(* IEC 61131-3 sources: Fischertechnik-RPi/Test, 12 files *)

(* ---- 1test.st ---- *)
PROGRAM Cell1
  VAR
    R1_front AT %IX0.2 : BOOL := true;
    R1_rear AT %IX0.3 : BOOL := true;
    C1_endIR AT %IX0.4 : BOOL := true;
    C1_startIR AT %IX0.5 : BOOL := true;
    Main AT %IX0.6 : BOOL := false;
    R1_fwd_motor AT %QX0.2 : BOOL := true;
    R1_bwd_motor AT %QX0.3 : BOOL := true;
    C1_motor AT %QX0.4 : BOOL := true;
  END_VAR
  VAR
    C1_working : BOOL := false;
    State1 : BOOL := false;
  END_VAR
  VAR
    State1_int AT %MD1 : DINT := 0;
  END_VAR
  VAR
    R1_in_transit : BOOL := false;
    State2 : BOOL := false;
  END_VAR
  VAR
    State2_int AT %MD3 : DINT := 0;
  END_VAR
  VAR
    R1_fwd : BOOL := false;
  END_VAR
  VAR
    R1_fwd_int AT %MD4 : DINT := 0;
  END_VAR
  VAR
    R1_bwd : BOOL := false;
  END_VAR
  VAR
    R1_bwd_int AT %MD5 : DINT := 0;
  END_VAR
  VAR
    Timer_in_transit : TON;
    BOOL_TO_DINT27_ENO : BOOL;
    BOOL_TO_DINT27_OUT : DINT;
    BOOL_TO_DINT37_ENO : BOOL;
    BOOL_TO_DINT37_OUT : DINT;
    BOOL_TO_DINT61_ENO : BOOL;
    BOOL_TO_DINT61_OUT : DINT;
    BOOL_TO_DINT67_ENO : BOOL;
    BOOL_TO_DINT67_OUT : DINT;
  END_VAR

  IF NOT(C1_startIR) THEN
    C1_working := TRUE; (*set*)
  END_IF;
  C1_motor := NOT(C1_working AND NOT(Main));
  IF C1_working AND NOT(C1_endIR) THEN
    R1_in_transit := TRUE; (*set*)
  END_IF;
  Timer_in_transit(IN := R1_in_transit AND C1_working, PT := T#1000ms);
  IF Timer_in_transit.Q THEN
    R1_fwd := TRUE; (*set*)
  END_IF;
  IF Timer_in_transit.Q THEN
    C1_working := FALSE; (*reset*)
  END_IF;
  IF Timer_in_transit.Q THEN
    R1_in_transit := FALSE; (*reset*)
  END_IF;
  R1_fwd_motor := NOT(R1_fwd AND NOT(Main));
  IF NOT(R1_front) AND R1_fwd THEN
    R1_bwd := TRUE; (*set*)
  END_IF;
  IF NOT(R1_front) AND R1_fwd THEN
    R1_fwd := FALSE; (*reset*)
  END_IF;
  R1_bwd_motor := NOT(R1_bwd AND NOT(Main));
  IF NOT(R1_rear) AND R1_bwd THEN
    R1_bwd := FALSE; (*reset*)
  END_IF;
  IF R1_in_transit AND C1_working THEN
    State1 := FALSE; (*reset*)
  END_IF;
  IF R1_in_transit AND C1_working THEN
    State2 := TRUE; (*set*)
  END_IF;
  IF NOT(R1_in_transit) AND C1_working THEN
    State1 := TRUE; (*set*)
  END_IF;
  IF NOT(R1_in_transit) AND NOT(C1_working) THEN
    State2 := FALSE; (*reset*)
  END_IF;
  BOOL_TO_DINT27_OUT := BOOL_TO_DINT(EN := TRUE, IN := State1, ENO => BOOL_TO_DINT27_ENO);
  State1_int := BOOL_TO_DINT27_OUT;
  BOOL_TO_DINT37_OUT := BOOL_TO_DINT(EN := TRUE, IN := State2, ENO => BOOL_TO_DINT37_ENO);
  State2_int := BOOL_TO_DINT37_OUT;
  BOOL_TO_DINT61_OUT := BOOL_TO_DINT(EN := TRUE, IN := R1_fwd, ENO => BOOL_TO_DINT61_ENO);
  R1_fwd_int := BOOL_TO_DINT61_OUT;
  BOOL_TO_DINT67_OUT := BOOL_TO_DINT(EN := TRUE, IN := R1_bwd, ENO => BOOL_TO_DINT67_ENO);
  R1_bwd_int := BOOL_TO_DINT67_OUT;
END_PROGRAM

CONFIGURATION Config0

  RESOURCE Res0 ON PLC
    TASK TaskMain(INTERVAL := T#50ms,PRIORITY := 0);
    PROGRAM Inst0 WITH TaskMain : Cell1;
  END_RESOURCE
END_CONFIGURATION

(* ---- FT_con02.st ---- *)
PROGRAM Cell2
  VAR
    C1_IR AT %IX0.3 : BOOL := true;
    M1_IR AT %IX0.4 : BOOL := true;
    Main AT %IX0.6 : BOOL := true;
    M1_motor AT %QX0.2 : BOOL := true;
    C2_motor AT %QX0.4 : BOOL := true;
  END_VAR
  VAR
    C2_working : BOOL := false;
  END_VAR
  VAR
    C2_working_int AT %MD1 : DINT := 0;
  END_VAR
  VAR
    C2_afterM : BOOL := false;
  END_VAR
  VAR
    C2_afterM_int AT %MD2 : DINT := 0;
  END_VAR
  VAR
    Step1 : BOOL := false;
  END_VAR
  VAR
    Step1_int AT %MD3 : DINT := 0;
  END_VAR
  VAR
    Step2 : BOOL := false;
  END_VAR
  VAR
    Step2_int AT %MD4 : DINT := 0;
  END_VAR
  VAR
    Step3 : BOOL := false;
  END_VAR
  VAR
    Step3_int AT %MD5 : DINT := 0;
  END_VAR
  VAR
    Pause1 : BOOL := false;
  END_VAR
  VAR
    Pause1_int AT %MD6 : DINT := 0;
  END_VAR
  VAR
    Pause2 : BOOL := false;
  END_VAR
  VAR
    Pause2_int AT %MD7 : DINT := 0;
  END_VAR
  VAR
    Timer_conveyor : TON;
    Timer_machining : TON;
    TON0 : TON;
    TON1 : TON;
    TON2 : TON;
    TON3 : TON;
    TON4 : TON;
    BOOL_TO_DINT41_ENO : BOOL;
    BOOL_TO_DINT41_OUT : DINT;
    BOOL_TO_DINT105_ENO : BOOL;
    BOOL_TO_DINT105_OUT : DINT;
    BOOL_TO_DINT51_ENO : BOOL;
    BOOL_TO_DINT51_OUT : DINT;
    BOOL_TO_DINT85_ENO : BOOL;
    BOOL_TO_DINT85_OUT : DINT;
    BOOL_TO_DINT90_ENO : BOOL;
    BOOL_TO_DINT90_OUT : DINT;
    BOOL_TO_DINT95_ENO : BOOL;
    BOOL_TO_DINT95_OUT : DINT;
    BOOL_TO_DINT100_ENO : BOOL;
    BOOL_TO_DINT100_OUT : DINT;
  END_VAR

  IF NOT(C1_IR) THEN
    C2_working := TRUE; (*set*)
  END_IF;
  C2_motor := NOT((C2_afterM OR C2_working) AND NOT(Main));
  IF NOT(M1_IR) AND C2_working THEN
    Step1 := TRUE; (*set*)
  END_IF;
  IF NOT(M1_IR) AND C2_working THEN
    C2_working := FALSE; (*reset*)
  END_IF;
  M1_motor := NOT((Step1 OR Step2 OR Step3) AND NOT(Main));
  TON0(IN := Step1, PT := T#1000ms);
  IF TON0.Q THEN
    Pause1 := TRUE; (*set*)
  END_IF;
  IF TON0.Q THEN
    Step1 := FALSE; (*reset*)
  END_IF;
  TON1(IN := Pause1, PT := T#1000ms);
  IF TON1.Q THEN
    Pause1 := FALSE; (*reset*)
  END_IF;
  IF TON1.Q THEN
    Step2 := TRUE; (*set*)
  END_IF;
  TON2(IN := Step2, PT := T#1000ms);
  IF TON2.Q THEN
    Pause2 := TRUE; (*set*)
  END_IF;
  IF TON2.Q THEN
    Step2 := FALSE; (*reset*)
  END_IF;
  TON3(IN := Pause2, PT := T#1000ms);
  IF TON3.Q THEN
    Pause2 := FALSE; (*reset*)
  END_IF;
  IF TON3.Q THEN
    Step3 := TRUE; (*set*)
  END_IF;
  Timer_machining(IN := Step3, PT := T#1000ms);
  IF Timer_machining.Q THEN
    C2_afterM := TRUE; (*set*)
  END_IF;
  IF Timer_machining.Q THEN
    Step3 := FALSE; (*reset*)
  END_IF;
  Timer_conveyor(IN := C2_working, PT := T#6000ms);
  IF Timer_conveyor.Q THEN
    C2_working := FALSE; (*reset*)
  END_IF;
  TON4(IN := C2_afterM, PT := T#2000ms);
  IF TON4.Q THEN
    C2_afterM := FALSE; (*reset*)
  END_IF;
  BOOL_TO_DINT41_OUT := BOOL_TO_DINT(EN := TRUE, IN := C2_working, ENO => BOOL_TO_DINT41_ENO);
  C2_working_int := BOOL_TO_DINT41_OUT;
  BOOL_TO_DINT105_OUT := BOOL_TO_DINT(EN := TRUE, IN := C2_afterM, ENO => BOOL_TO_DINT105_ENO);
  C2_afterM_int := BOOL_TO_DINT105_OUT;
  BOOL_TO_DINT51_OUT := BOOL_TO_DINT(EN := TRUE, IN := Step1, ENO => BOOL_TO_DINT51_ENO);
  Step1_int := BOOL_TO_DINT51_OUT;
  BOOL_TO_DINT85_OUT := BOOL_TO_DINT(EN := TRUE, IN := Step2, ENO => BOOL_TO_DINT85_ENO);
  Step2_int := BOOL_TO_DINT85_OUT;
  BOOL_TO_DINT90_OUT := BOOL_TO_DINT(EN := TRUE, IN := Step3, ENO => BOOL_TO_DINT90_ENO);
  Step3_int := BOOL_TO_DINT90_OUT;
  BOOL_TO_DINT95_OUT := BOOL_TO_DINT(EN := TRUE, IN := Pause1, ENO => BOOL_TO_DINT95_ENO);
  Pause1_int := BOOL_TO_DINT95_OUT;
  BOOL_TO_DINT100_OUT := BOOL_TO_DINT(EN := TRUE, IN := Pause2, ENO => BOOL_TO_DINT100_ENO);
  Pause2_int := BOOL_TO_DINT100_OUT;
END_PROGRAM

CONFIGURATION Config0

  RESOURCE Res0 ON PLC
    TASK TaskMain(INTERVAL := T#50ms,PRIORITY := 0);
    PROGRAM Inst0 WITH TaskMain : Cell2;
  END_RESOURCE
END_CONFIGURATION

(* ---- FT_con03.st ---- *)
PROGRAM Cell3
  VAR
    C2_IR AT %IX0.3 : BOOL := true;
    M2_IR AT %IX0.4 : BOOL := true;
    Main AT %IX0.6 : BOOL := true;
    M2_motor AT %QX0.2 : BOOL := true;
    C3_motor AT %QX0.4 : BOOL := true;
  END_VAR
  VAR
    C3_working : BOOL := false;
  END_VAR
  VAR
    C3_working_int AT %MD1 : DINT := 0;
  END_VAR
  VAR
    C3_afterM : BOOL := false;
  END_VAR
  VAR
    C3_afterM_int AT %MD2 : DINT := 0;
  END_VAR
  VAR
    Step1 : BOOL := false;
  END_VAR
  VAR
    Step1_int AT %MD3 : DINT := 0;
  END_VAR
  VAR
    Step2 : BOOL := false;
  END_VAR
  VAR
    Step2_int AT %MD4 : DINT := 0;
  END_VAR
  VAR
    Pause : BOOL := false;
  END_VAR
  VAR
    Pause_int AT %MD5 : DINT := 0;
  END_VAR
  VAR
    Timer_conveyor : TON;
    Timer_machining : TON;
    TON0 : TON;
    TON1 : TON;
    TON2 : TON;
    TON3 : TON;
    BOOL_TO_DINT70_ENO : BOOL;
    BOOL_TO_DINT70_OUT : DINT;
    BOOL_TO_DINT41_ENO : BOOL;
    BOOL_TO_DINT41_OUT : DINT;
    BOOL_TO_DINT51_ENO : BOOL;
    BOOL_TO_DINT51_OUT : DINT;
    BOOL_TO_DINT75_ENO : BOOL;
    BOOL_TO_DINT75_OUT : DINT;
    BOOL_TO_DINT80_ENO : BOOL;
    BOOL_TO_DINT80_OUT : DINT;
  END_VAR

  TON0(IN := NOT(C2_IR), PT := T#5000ms);
  IF TON0.Q THEN
    C3_working := TRUE; (*set*)
  END_IF;
  C3_motor := NOT((C3_afterM OR C3_working) AND NOT(Main));
  IF NOT(M2_IR) AND C3_working THEN
    Step1 := TRUE; (*set*)
  END_IF;
  IF NOT(M2_IR) AND C3_working THEN
    C3_working := FALSE; (*reset*)
  END_IF;
  M2_motor := NOT((Step1 OR Step2) AND NOT(Main));
  Timer_machining(IN := Step1, PT := T#2000ms);
  IF Timer_machining.Q THEN
    Pause := TRUE; (*set*)
  END_IF;
  IF Timer_machining.Q THEN
    Step1 := FALSE; (*reset*)
  END_IF;
  TON2(IN := Pause, PT := T#1000ms);
  IF TON2.Q THEN
    Step2 := TRUE; (*set*)
  END_IF;
  IF TON2.Q THEN
    Pause := FALSE; (*reset*)
  END_IF;
  TON1(IN := Step2, PT := T#2000ms);
  IF TON1.Q THEN
    C3_afterM := TRUE; (*set*)
  END_IF;
  IF TON1.Q THEN
    Step2 := FALSE; (*reset*)
  END_IF;
  Timer_conveyor(IN := C3_working, PT := T#6000ms);
  IF Timer_conveyor.Q THEN
    C3_working := FALSE; (*reset*)
  END_IF;
  TON3(IN := C3_afterM, PT := T#3000ms);
  IF TON3.Q THEN
    C3_afterM := FALSE; (*reset*)
  END_IF;
  BOOL_TO_DINT70_OUT := BOOL_TO_DINT(EN := TRUE, IN := C3_working, ENO => BOOL_TO_DINT70_ENO);
  C3_working_int := BOOL_TO_DINT70_OUT;
  BOOL_TO_DINT41_OUT := BOOL_TO_DINT(EN := TRUE, IN := C3_afterM, ENO => BOOL_TO_DINT41_ENO);
  C3_afterM_int := BOOL_TO_DINT41_OUT;
  BOOL_TO_DINT51_OUT := BOOL_TO_DINT(EN := TRUE, IN := Step1, ENO => BOOL_TO_DINT51_ENO);
  Step1_int := BOOL_TO_DINT51_OUT;
  BOOL_TO_DINT75_OUT := BOOL_TO_DINT(EN := TRUE, IN := Step2, ENO => BOOL_TO_DINT75_ENO);
  Step2_int := BOOL_TO_DINT75_OUT;
  BOOL_TO_DINT80_OUT := BOOL_TO_DINT(EN := TRUE, IN := Pause, ENO => BOOL_TO_DINT80_ENO);
  Pause_int := BOOL_TO_DINT80_OUT;
END_PROGRAM

CONFIGURATION Config0

  RESOURCE Res0 ON PLC
    TASK TaskMain(INTERVAL := T#50ms,PRIORITY := 0);
    PROGRAM Inst0 WITH TaskMain : Cell3;
  END_RESOURCE
END_CONFIGURATION

(* ---- FT_con04.st ---- *)
PROGRAM Cell4
  VAR
    R2_front AT %IX0.2 : BOOL := true;
    R2_rear AT %IX0.3 : BOOL := true;
    C4_endIR AT %IX0.4 : BOOL := true;
    C3_IR AT %IX0.5 : BOOL := true;
    Main AT %IX0.6 : BOOL := false;
    R2_fwd_motor AT %QX0.2 : BOOL := true;
    R2_bwd_motor AT %QX0.3 : BOOL := true;
    C4_motor AT %QX0.4 : BOOL := true;
  END_VAR
  VAR
    C4_working : BOOL := false;
  END_VAR
  VAR
    C4_working_int AT %MD1 : DINT := 0;
  END_VAR
  VAR
    R2_in_transit : BOOL := false;
  END_VAR
  VAR
    R2_in_transit_int AT %MD3 : DINT := 0;
  END_VAR
  VAR
    R2_fwd : BOOL := false;
  END_VAR
  VAR
    R2_fwd_int AT %MD4 : DINT := 0;
  END_VAR
  VAR
    R2_bwd : BOOL := false;
  END_VAR
  VAR
    R2_bwd_int AT %MD5 : DINT := 0;
  END_VAR
  VAR
    Timer_in_transit : TON;
    BOOL_TO_DINT49_ENO : BOOL;
    BOOL_TO_DINT49_OUT : DINT;
    BOOL_TO_DINT64_ENO : BOOL;
    BOOL_TO_DINT64_OUT : DINT;
    BOOL_TO_DINT61_ENO : BOOL;
    BOOL_TO_DINT61_OUT : DINT;
    BOOL_TO_DINT67_ENO : BOOL;
    BOOL_TO_DINT67_OUT : DINT;
  END_VAR

  IF NOT(C3_IR) THEN
    R2_in_transit := TRUE; (*set*)
  END_IF;
  Timer_in_transit(IN := R2_in_transit, PT := T#6000ms);
  IF Timer_in_transit.Q THEN
    R2_fwd := TRUE; (*set*)
  END_IF;
  IF Timer_in_transit.Q THEN
    C4_working := TRUE; (*set*)
  END_IF;
  IF Timer_in_transit.Q THEN
    R2_in_transit := FALSE; (*reset*)
  END_IF;
  R2_fwd_motor := NOT(R2_fwd AND NOT(Main));
  IF NOT(R2_front) AND R2_fwd THEN
    R2_bwd := TRUE; (*set*)
  END_IF;
  IF NOT(R2_front) AND R2_fwd THEN
    R2_fwd := FALSE; (*reset*)
  END_IF;
  R2_bwd_motor := NOT(R2_bwd AND NOT(Main) AND TRUE);
  IF NOT(R2_rear) AND R2_bwd THEN
    R2_bwd := FALSE; (*reset*)
  END_IF;
  C4_motor := NOT(C4_working AND NOT(Main));
  IF NOT(C4_endIR) AND C4_working THEN
    C4_working := FALSE; (*reset*)
  END_IF;
  BOOL_TO_DINT49_OUT := BOOL_TO_DINT(EN := TRUE, IN := C4_working, ENO => BOOL_TO_DINT49_ENO);
  C4_working_int := BOOL_TO_DINT49_OUT;
  BOOL_TO_DINT64_OUT := BOOL_TO_DINT(EN := TRUE, IN := R2_in_transit, ENO => BOOL_TO_DINT64_ENO);
  R2_in_transit_int := BOOL_TO_DINT64_OUT;
  BOOL_TO_DINT61_OUT := BOOL_TO_DINT(EN := TRUE, IN := R2_fwd, ENO => BOOL_TO_DINT61_ENO);
  R2_fwd_int := BOOL_TO_DINT61_OUT;
  BOOL_TO_DINT67_OUT := BOOL_TO_DINT(EN := TRUE, IN := R2_bwd, ENO => BOOL_TO_DINT67_ENO);
  R2_bwd_int := BOOL_TO_DINT67_OUT;
END_PROGRAM

CONFIGURATION Config0

  RESOURCE Res0 ON PLC
    TASK TaskMain(INTERVAL := T#50ms,PRIORITY := 0);
    PROGRAM Inst0 WITH TaskMain : Cell4;
  END_RESOURCE
END_CONFIGURATION

(* ---- FT_con04b.st ---- *)
PROGRAM Cell4
  VAR
    R2_front AT %IX0.2 : BOOL := true;
    R2_rear AT %IX0.3 : BOOL := true;
    C4_endIR AT %IX0.4 : BOOL := true;
    C3_IR AT %IX0.5 : BOOL := true;
    Main AT %IX0.6 : BOOL := false;
    R2_fwd_motor AT %QX0.2 : BOOL := true;
    R2_bwd_motor AT %QX0.3 : BOOL := true;
    C4_motor AT %QX0.4 : BOOL := true;
  END_VAR
  VAR
    C4_working : BOOL := false;
    C4_R2f : BOOL := false;
  END_VAR
  VAR
    C4_R2f_int AT %MD1 : DINT := 0;
  END_VAR
  VAR
    R2_in_transit : BOOL := false;
  END_VAR
  VAR
    R2_in_transit_int AT %MD3 : DINT := 0;
  END_VAR
  VAR
    R2_fwd : BOOL := false;
    C4_R2b : BOOL := false;
  END_VAR
  VAR
    C4_R2b_int AT %MD4 : DINT := 0;
  END_VAR
  VAR
    R2_bwd : BOOL := false;
    R2b_solo : BOOL := false;
  END_VAR
  VAR
    R2b_solo_int AT %MD5 : DINT := 0;
  END_VAR
  VAR
    Timer_in_transit : TON;
    BOOL_TO_DINT49_ENO : BOOL;
    BOOL_TO_DINT49_OUT : DINT;
    BOOL_TO_DINT64_ENO : BOOL;
    BOOL_TO_DINT64_OUT : DINT;
    BOOL_TO_DINT61_ENO : BOOL;
    BOOL_TO_DINT61_OUT : DINT;
    BOOL_TO_DINT67_ENO : BOOL;
    BOOL_TO_DINT67_OUT : DINT;
  END_VAR

  IF NOT(C3_IR) THEN
    R2_in_transit := TRUE; (*set*)
  END_IF;
  Timer_in_transit(IN := R2_in_transit, PT := T#6000ms);
  IF Timer_in_transit.Q THEN
    R2_fwd := TRUE; (*set*)
  END_IF;
  IF Timer_in_transit.Q THEN
    C4_working := TRUE; (*set*)
  END_IF;
  IF Timer_in_transit.Q THEN
    R2_in_transit := FALSE; (*reset*)
  END_IF;
  R2_fwd_motor := NOT(R2_fwd AND NOT(Main));
  IF NOT(R2_front) AND R2_fwd THEN
    R2_bwd := TRUE; (*set*)
  END_IF;
  IF NOT(R2_front) AND R2_fwd THEN
    R2_fwd := FALSE; (*reset*)
  END_IF;
  R2_bwd_motor := NOT(R2_bwd AND NOT(Main) AND TRUE);
  IF NOT(R2_rear) AND R2_bwd THEN
    R2_bwd := FALSE; (*reset*)
  END_IF;
  IF NOT(R2_bwd) THEN
    R2b_solo := FALSE; (*reset*)
  END_IF;
  C4_motor := NOT(C4_working AND NOT(Main));
  IF NOT(C4_endIR) AND C4_working THEN
    C4_working := FALSE; (*reset*)
  END_IF;
  IF R2_fwd AND C4_working THEN
    C4_R2f := TRUE; (*set*)
  END_IF;
  IF R2_bwd AND C4_working THEN
    C4_R2b := TRUE; (*set*)
  END_IF;
  IF R2_fwd AND C4_working THEN
    C4_R2f := TRUE; (*set*)
  END_IF;
  IF R2_fwd AND C4_working THEN
    C4_R2f := TRUE; (*set*)
  END_IF;
  IF R2_bwd AND C4_working THEN
    C4_R2f := FALSE; (*reset*)
  END_IF;
  IF C4_R2b AND NOT(C4_working) THEN
    R2b_solo := TRUE; (*set*)
  END_IF;
  IF C4_R2b AND NOT(C4_working) THEN
    C4_R2b := FALSE; (*reset*)
  END_IF;
  BOOL_TO_DINT49_OUT := BOOL_TO_DINT(EN := TRUE, IN := C4_R2f, ENO => BOOL_TO_DINT49_ENO);
  C4_R2f_int := BOOL_TO_DINT49_OUT;
  BOOL_TO_DINT64_OUT := BOOL_TO_DINT(EN := TRUE, IN := R2_in_transit, ENO => BOOL_TO_DINT64_ENO);
  R2_in_transit_int := BOOL_TO_DINT64_OUT;
  BOOL_TO_DINT61_OUT := BOOL_TO_DINT(EN := TRUE, IN := C4_R2b, ENO => BOOL_TO_DINT61_ENO);
  C4_R2b_int := BOOL_TO_DINT61_OUT;
  BOOL_TO_DINT67_OUT := BOOL_TO_DINT(EN := TRUE, IN := R2b_solo, ENO => BOOL_TO_DINT67_ENO);
  R2b_solo_int := BOOL_TO_DINT67_OUT;
END_PROGRAM

CONFIGURATION Config0

  RESOURCE Res0 ON PLC
    TASK TaskMain(INTERVAL := T#50ms,PRIORITY := 0);
    PROGRAM Inst0 WITH TaskMain : Cell4;
  END_RESOURCE
END_CONFIGURATION

(* ---- scratch4.st ---- *)
PROGRAM Cell4
  VAR
    R2_front AT %IX0.2 : BOOL := true;
  END_VAR
  VAR
    C3_IR_working : BOOL := false;
  END_VAR
  VAR
    R2_rear AT %IX0.3 : BOOL := true;
    C4_endIR AT %IX0.4 : BOOL := true;
    C3_IR AT %IX0.5 : BOOL := true;
    Main AT %IX0.6 : BOOL := false;
    R2_fwd_motor AT %QX0.2 : BOOL := true;
    R2_bwd_motor AT %QX0.3 : BOOL := true;
    C4_motor AT %QX0.4 : BOOL := true;
  END_VAR
  VAR
    C4_working : BOOL := false;
  END_VAR
  VAR
    C4_working_int AT %MD1 : DINT := 0;
  END_VAR
  VAR
    R2_in_transit : BOOL := false;
  END_VAR
  VAR
    R2_in_transit_int AT %MD3 : DINT := 0;
  END_VAR
  VAR
    R2_fwd : BOOL := false;
  END_VAR
  VAR
    R2_fwd_int AT %MD4 : DINT := 0;
  END_VAR
  VAR
    R2_bwd : BOOL := false;
  END_VAR
  VAR
    R2_bwd_int AT %MD5 : DINT := 0;
  END_VAR
  VAR
    Timer_in_transit : TON;
  END_VAR
  VAR
    Scratch AT %QX0.7 : BOOL := false;
  END_VAR
  VAR
    BOOL_TO_DINT49_ENO : BOOL;
    BOOL_TO_DINT49_OUT : DINT;
    BOOL_TO_DINT64_ENO : BOOL;
    BOOL_TO_DINT64_OUT : DINT;
    BOOL_TO_DINT61_ENO : BOOL;
    BOOL_TO_DINT61_OUT : DINT;
    BOOL_TO_DINT67_ENO : BOOL;
    BOOL_TO_DINT67_OUT : DINT;
  END_VAR

  Timer_in_transit(IN := Scratch, PT := T#1000ms);
  IF Timer_in_transit.Q THEN
    R2_fwd := TRUE; (*set*)
  END_IF;
  IF Timer_in_transit.Q THEN
    C4_working := TRUE; (*set*)
  END_IF;
  IF Timer_in_transit.Q THEN
    R2_in_transit := FALSE; (*reset*)
  END_IF;
  R2_fwd_motor := NOT(R2_fwd AND NOT(Main));
  IF Timer_in_transit.Q THEN
    C3_IR_working := FALSE; (*reset*)
  END_IF;
  IF NOT(R2_front) AND R2_fwd THEN
    R2_bwd := TRUE; (*set*)
  END_IF;
  IF NOT(R2_front) AND R2_fwd THEN
    R2_fwd := FALSE; (*reset*)
  END_IF;
  R2_bwd_motor := NOT(R2_bwd AND NOT(Main) AND TRUE);
  IF NOT(R2_rear) AND R2_bwd THEN
    R2_bwd := FALSE; (*reset*)
  END_IF;
  C4_motor := NOT(C4_working AND NOT(Main));
  IF NOT(C4_endIR) AND C4_working THEN
    C4_working := FALSE; (*reset*)
  END_IF;
  BOOL_TO_DINT49_OUT := BOOL_TO_DINT(EN := TRUE, IN := C4_working, ENO => BOOL_TO_DINT49_ENO);
  C4_working_int := BOOL_TO_DINT49_OUT;
  BOOL_TO_DINT64_OUT := BOOL_TO_DINT(EN := TRUE, IN := R2_in_transit, ENO => BOOL_TO_DINT64_ENO);
  R2_in_transit_int := BOOL_TO_DINT64_OUT;
  BOOL_TO_DINT61_OUT := BOOL_TO_DINT(EN := TRUE, IN := R2_fwd, ENO => BOOL_TO_DINT61_ENO);
  R2_fwd_int := BOOL_TO_DINT61_OUT;
  BOOL_TO_DINT67_OUT := BOOL_TO_DINT(EN := TRUE, IN := R2_bwd, ENO => BOOL_TO_DINT67_ENO);
  R2_bwd_int := BOOL_TO_DINT67_OUT;
END_PROGRAM

CONFIGURATION Config0

  RESOURCE Res0 ON PLC
    TASK TaskMain(INTERVAL := T#50ms,PRIORITY := 0);
    PROGRAM Inst0 WITH TaskMain : Cell4;
  END_RESOURCE
END_CONFIGURATION

(* ---- scratch42.st ---- *)
PROGRAM Cell4
  VAR
    R2_front AT %IX0.2 : BOOL := true;
  END_VAR
  VAR
    C3_IR_working : BOOL := false;
  END_VAR
  VAR
    R2_rear AT %IX0.3 : BOOL := true;
    C4_endIR AT %IX0.4 : BOOL := true;
    C3_IR AT %IX0.5 : BOOL := true;
    Main AT %IX0.6 : BOOL := false;
    R2_fwd_motor AT %QX0.2 : BOOL := true;
    R2_bwd_motor AT %QX0.3 : BOOL := true;
    C4_motor AT %QX0.4 : BOOL := true;
  END_VAR
  VAR
    C4_working : BOOL := false;
  END_VAR
  VAR
    C4_working_int AT %MD1 : DINT := 0;
  END_VAR
  VAR
    R2_in_transit : BOOL := false;
  END_VAR
  VAR
    R2_in_transit_int AT %MD3 : DINT := 0;
  END_VAR
  VAR
    R2_fwd : BOOL := false;
  END_VAR
  VAR
    R2_fwd_int AT %MD4 : DINT := 0;
  END_VAR
  VAR
    R2_bwd : BOOL := false;
  END_VAR
  VAR
    R2_bwd_int AT %MD5 : DINT := 0;
  END_VAR
  VAR
    Timer_in_transit : TON;
  END_VAR
  VAR
    Scratch AT %QX0.7 : BOOL := true;
  END_VAR
  VAR
    BOOL_TO_DINT49_ENO : BOOL;
    BOOL_TO_DINT49_OUT : DINT;
    BOOL_TO_DINT64_ENO : BOOL;
    BOOL_TO_DINT64_OUT : DINT;
    BOOL_TO_DINT61_ENO : BOOL;
    BOOL_TO_DINT61_OUT : DINT;
    BOOL_TO_DINT67_ENO : BOOL;
    BOOL_TO_DINT67_OUT : DINT;
  END_VAR

  Timer_in_transit(IN := NOT(Scratch), PT := T#1000ms);
  IF Timer_in_transit.Q THEN
    R2_fwd := TRUE; (*set*)
  END_IF;
  IF Timer_in_transit.Q THEN
    C4_working := TRUE; (*set*)
  END_IF;
  IF Timer_in_transit.Q THEN
    R2_in_transit := FALSE; (*reset*)
  END_IF;
  R2_fwd_motor := NOT(R2_fwd AND NOT(Main));
  IF Timer_in_transit.Q THEN
    C3_IR_working := FALSE; (*reset*)
  END_IF;
  IF NOT(R2_front) AND R2_fwd THEN
    R2_bwd := TRUE; (*set*)
  END_IF;
  IF NOT(R2_front) AND R2_fwd THEN
    R2_fwd := FALSE; (*reset*)
  END_IF;
  R2_bwd_motor := NOT(R2_bwd AND NOT(Main) AND TRUE);
  IF NOT(R2_rear) AND R2_bwd THEN
    R2_bwd := FALSE; (*reset*)
  END_IF;
  C4_motor := NOT(C4_working AND NOT(Main));
  IF NOT(C4_endIR) AND C4_working THEN
    C4_working := FALSE; (*reset*)
  END_IF;
  BOOL_TO_DINT49_OUT := BOOL_TO_DINT(EN := TRUE, IN := C4_working, ENO => BOOL_TO_DINT49_ENO);
  C4_working_int := BOOL_TO_DINT49_OUT;
  BOOL_TO_DINT64_OUT := BOOL_TO_DINT(EN := TRUE, IN := R2_in_transit, ENO => BOOL_TO_DINT64_ENO);
  R2_in_transit_int := BOOL_TO_DINT64_OUT;
  BOOL_TO_DINT61_OUT := BOOL_TO_DINT(EN := TRUE, IN := R2_fwd, ENO => BOOL_TO_DINT61_ENO);
  R2_fwd_int := BOOL_TO_DINT61_OUT;
  BOOL_TO_DINT67_OUT := BOOL_TO_DINT(EN := TRUE, IN := R2_bwd, ENO => BOOL_TO_DINT67_ENO);
  R2_bwd_int := BOOL_TO_DINT67_OUT;
END_PROGRAM

CONFIGURATION Config0

  RESOURCE Res0 ON PLC
    TASK TaskMain(INTERVAL := T#50ms,PRIORITY := 0);
    PROGRAM Inst0 WITH TaskMain : Cell4;
  END_RESOURCE
END_CONFIGURATION

(* ---- scratch420.st ---- *)
PROGRAM Cell4
  VAR
    R2_front AT %IX0.2 : BOOL := true;
  END_VAR
  VAR
    C3_IR_working : BOOL := false;
  END_VAR
  VAR
    R2_rear AT %IX0.3 : BOOL := true;
    C4_endIR AT %IX0.4 : BOOL := true;
    Main AT %IX0.6 : BOOL := false;
    R2_fwd_motor AT %QX0.2 : BOOL := true;
    R2_bwd_motor AT %QX0.3 : BOOL := true;
    C4_motor AT %QX0.4 : BOOL := true;
  END_VAR
  VAR
    C4_working : BOOL := false;
  END_VAR
  VAR
    C4_working_int AT %MD1 : DINT := 0;
  END_VAR
  VAR
    R2_in_transit : BOOL := false;
  END_VAR
  VAR
    R2_in_transit_int AT %MD3 : DINT := 0;
  END_VAR
  VAR
    R2_fwd : BOOL := false;
  END_VAR
  VAR
    R2_fwd_int AT %MD4 : DINT := 0;
  END_VAR
  VAR
    R2_bwd : BOOL := false;
  END_VAR
  VAR
    R2_bwd_int AT %MD5 : DINT := 0;
  END_VAR
  VAR
    Timer_in_transit : TON;
  END_VAR
  VAR
    Scratch AT %QX0.7 : BOOL := true;
  END_VAR
  VAR
    BOOL_TO_DINT49_ENO : BOOL;
    BOOL_TO_DINT49_OUT : DINT;
    BOOL_TO_DINT64_ENO : BOOL;
    BOOL_TO_DINT64_OUT : DINT;
    BOOL_TO_DINT61_ENO : BOOL;
    BOOL_TO_DINT61_OUT : DINT;
    BOOL_TO_DINT67_ENO : BOOL;
    BOOL_TO_DINT67_OUT : DINT;
  END_VAR

  Timer_in_transit(IN := NOT(Scratch), PT := T#1000ms);
  IF Timer_in_transit.Q THEN
    R2_fwd := TRUE; (*set*)
  END_IF;
  IF Timer_in_transit.Q THEN
    C4_working := TRUE; (*set*)
  END_IF;
  IF Timer_in_transit.Q THEN
    R2_in_transit := FALSE; (*reset*)
  END_IF;
  R2_fwd_motor := NOT(R2_fwd AND NOT(Main));
  IF Timer_in_transit.Q THEN
    C3_IR_working := FALSE; (*reset*)
  END_IF;
  IF NOT(R2_front) AND R2_fwd THEN
    R2_bwd := TRUE; (*set*)
  END_IF;
  IF NOT(R2_front) AND R2_fwd THEN
    R2_fwd := FALSE; (*reset*)
  END_IF;
  R2_bwd_motor := NOT(R2_bwd AND NOT(Main) AND TRUE);
  IF NOT(R2_rear) AND R2_bwd THEN
    R2_bwd := FALSE; (*reset*)
  END_IF;
  C4_motor := NOT(C4_working AND NOT(Main));
  IF NOT(C4_endIR) AND C4_working THEN
    C4_working := FALSE; (*reset*)
  END_IF;
  BOOL_TO_DINT49_OUT := BOOL_TO_DINT(EN := TRUE, IN := C4_working, ENO => BOOL_TO_DINT49_ENO);
  C4_working_int := BOOL_TO_DINT49_OUT;
  BOOL_TO_DINT64_OUT := BOOL_TO_DINT(EN := TRUE, IN := R2_in_transit, ENO => BOOL_TO_DINT64_ENO);
  R2_in_transit_int := BOOL_TO_DINT64_OUT;
  BOOL_TO_DINT61_OUT := BOOL_TO_DINT(EN := TRUE, IN := R2_fwd, ENO => BOOL_TO_DINT61_ENO);
  R2_fwd_int := BOOL_TO_DINT61_OUT;
  BOOL_TO_DINT67_OUT := BOOL_TO_DINT(EN := TRUE, IN := R2_bwd, ENO => BOOL_TO_DINT67_ENO);
  R2_bwd_int := BOOL_TO_DINT67_OUT;
END_PROGRAM

CONFIGURATION Config0

  RESOURCE Res0 ON PLC
    TASK TaskMain(INTERVAL := T#50ms,PRIORITY := 0);
    PROGRAM Inst0 WITH TaskMain : Cell4;
  END_RESOURCE
END_CONFIGURATION

(* ---- scratch4201.st ---- *)
PROGRAM Cell4
  VAR
    R2_front AT %IX0.2 : BOOL := true;
  END_VAR
  VAR
    C3_IR_working : BOOL := false;
  END_VAR
  VAR
    R2_rear AT %IX0.3 : BOOL := true;
    C4_endIR AT %IX0.4 : BOOL := true;
    Main AT %IX0.6 : BOOL := false;
    R2_fwd_motor AT %QX0.2 : BOOL := true;
    R2_bwd_motor AT %QX0.3 : BOOL := true;
    C4_motor AT %QX0.4 : BOOL := true;
  END_VAR
  VAR
    C4_working : BOOL := false;
  END_VAR
  VAR
    C4_working_int AT %MD1 : DINT := 0;
  END_VAR
  VAR
    R2_in_transit : BOOL := false;
  END_VAR
  VAR
    R2_in_transit_int AT %MD3 : DINT := 0;
  END_VAR
  VAR
    R2_fwd : BOOL := false;
  END_VAR
  VAR
    R2_fwd_int AT %MD4 : DINT := 0;
  END_VAR
  VAR
    R2_bwd : BOOL := false;
  END_VAR
  VAR
    R2_bwd_int AT %MD5 : DINT := 0;
  END_VAR
  VAR
    Timer_in_transit : TON;
  END_VAR
  VAR
    Scratch AT %IX0.7 : BOOL := true;
  END_VAR
  VAR
    BOOL_TO_DINT49_ENO : BOOL;
    BOOL_TO_DINT49_OUT : DINT;
    BOOL_TO_DINT64_ENO : BOOL;
    BOOL_TO_DINT64_OUT : DINT;
    BOOL_TO_DINT61_ENO : BOOL;
    BOOL_TO_DINT61_OUT : DINT;
    BOOL_TO_DINT67_ENO : BOOL;
    BOOL_TO_DINT67_OUT : DINT;
  END_VAR

  Timer_in_transit(IN := NOT(Scratch), PT := T#1000ms);
  IF Timer_in_transit.Q THEN
    R2_fwd := TRUE; (*set*)
  END_IF;
  IF Timer_in_transit.Q THEN
    C4_working := TRUE; (*set*)
  END_IF;
  IF Timer_in_transit.Q THEN
    R2_in_transit := FALSE; (*reset*)
  END_IF;
  R2_fwd_motor := NOT(R2_fwd AND NOT(Main));
  IF Timer_in_transit.Q THEN
    C3_IR_working := FALSE; (*reset*)
  END_IF;
  IF NOT(R2_front) AND R2_fwd THEN
    R2_bwd := TRUE; (*set*)
  END_IF;
  IF NOT(R2_front) AND R2_fwd THEN
    R2_fwd := FALSE; (*reset*)
  END_IF;
  R2_bwd_motor := NOT(R2_bwd AND NOT(Main) AND TRUE);
  IF NOT(R2_rear) AND R2_bwd THEN
    R2_bwd := FALSE; (*reset*)
  END_IF;
  C4_motor := NOT(C4_working AND NOT(Main));
  IF NOT(C4_endIR) AND C4_working THEN
    C4_working := FALSE; (*reset*)
  END_IF;
  BOOL_TO_DINT49_OUT := BOOL_TO_DINT(EN := TRUE, IN := C4_working, ENO => BOOL_TO_DINT49_ENO);
  C4_working_int := BOOL_TO_DINT49_OUT;
  BOOL_TO_DINT64_OUT := BOOL_TO_DINT(EN := TRUE, IN := R2_in_transit, ENO => BOOL_TO_DINT64_ENO);
  R2_in_transit_int := BOOL_TO_DINT64_OUT;
  BOOL_TO_DINT61_OUT := BOOL_TO_DINT(EN := TRUE, IN := R2_fwd, ENO => BOOL_TO_DINT61_ENO);
  R2_fwd_int := BOOL_TO_DINT61_OUT;
  BOOL_TO_DINT67_OUT := BOOL_TO_DINT(EN := TRUE, IN := R2_bwd, ENO => BOOL_TO_DINT67_ENO);
  R2_bwd_int := BOOL_TO_DINT67_OUT;
END_PROGRAM

CONFIGURATION Config0

  RESOURCE Res0 ON PLC
    TASK TaskMain(INTERVAL := T#50ms,PRIORITY := 0);
    PROGRAM Inst0 WITH TaskMain : Cell4;
  END_RESOURCE
END_CONFIGURATION

(* ---- test2.st ---- *)
PROGRAM Cell2
  VAR
    C1_IR AT %IX0.3 : BOOL := true;
    M1_IR AT %IX0.4 : BOOL := true;
    Main AT %IX0.6 : BOOL := true;
    M1_motor AT %QX0.2 : BOOL := true;
    C2_motor AT %QX0.4 : BOOL := true;
  END_VAR
  VAR
    C2_working : BOOL := false;
  END_VAR
  VAR
    C2_working_int AT %MD1 : DINT := 0;
  END_VAR
  VAR
    C2_afterM : BOOL := false;
  END_VAR
  VAR
    C2_afterM_int AT %MD2 : DINT := 0;
  END_VAR
  VAR
    Step1 : BOOL := false;
  END_VAR
  VAR
    Step1_int AT %MD3 : DINT := 0;
  END_VAR
  VAR
    Step2 : BOOL := false;
  END_VAR
  VAR
    Step2_int AT %MD4 : DINT := 0;
  END_VAR
  VAR
    Step3 : BOOL := false;
  END_VAR
  VAR
    Step3_int AT %MD5 : DINT := 0;
  END_VAR
  VAR
    Pause1 : BOOL := false;
  END_VAR
  VAR
    Pause1_int AT %MD6 : DINT := 0;
  END_VAR
  VAR
    Pause2 : BOOL := false;
  END_VAR
  VAR
    Pause2_int AT %MD7 : DINT := 0;
  END_VAR
  VAR
    Timer_conveyor : TON;
    Timer_machining : TON;
    TON0 : TON;
    TON1 : TON;
    TON2 : TON;
    TON3 : TON;
    TON4 : TON;
    BOOL_TO_DINT41_ENO : BOOL;
    BOOL_TO_DINT41_OUT : DINT;
    BOOL_TO_DINT105_ENO : BOOL;
    BOOL_TO_DINT105_OUT : DINT;
    BOOL_TO_DINT51_ENO : BOOL;
    BOOL_TO_DINT51_OUT : DINT;
    BOOL_TO_DINT85_ENO : BOOL;
    BOOL_TO_DINT85_OUT : DINT;
    BOOL_TO_DINT90_ENO : BOOL;
    BOOL_TO_DINT90_OUT : DINT;
    BOOL_TO_DINT95_ENO : BOOL;
    BOOL_TO_DINT95_OUT : DINT;
    BOOL_TO_DINT100_ENO : BOOL;
    BOOL_TO_DINT100_OUT : DINT;
  END_VAR

  IF NOT(C1_IR) THEN
    C2_working := TRUE; (*set*)
  END_IF;
  C2_motor := NOT((C2_afterM OR C2_working) AND NOT(Main));
  IF NOT(M1_IR) AND C2_working THEN
    Step1 := TRUE; (*set*)
  END_IF;
  IF NOT(M1_IR) AND C2_working THEN
    C2_working := FALSE; (*reset*)
  END_IF;
  M1_motor := NOT((Step1 OR Step2 OR Step3) AND NOT(Main));
  TON0(IN := Step1, PT := T#1000ms);
  IF TON0.Q THEN
    Pause1 := TRUE; (*set*)
  END_IF;
  IF TON0.Q THEN
    Step1 := FALSE; (*reset*)
  END_IF;
  TON1(IN := Pause1, PT := T#1000ms);
  IF TON1.Q THEN
    Pause1 := FALSE; (*reset*)
  END_IF;
  IF TON1.Q THEN
    Step2 := TRUE; (*set*)
  END_IF;
  TON2(IN := Step2, PT := T#1000ms);
  IF TON2.Q THEN
    Pause2 := TRUE; (*set*)
  END_IF;
  IF TON2.Q THEN
    Step2 := FALSE; (*reset*)
  END_IF;
  TON3(IN := Pause2);
  IF TON3.Q THEN
    Pause2 := FALSE; (*reset*)
  END_IF;
  IF TON3.Q THEN
    Step3 := TRUE; (*set*)
  END_IF;
  Timer_machining(IN := Step3, PT := T#1000ms);
  IF Timer_machining.Q THEN
    C2_afterM := TRUE; (*set*)
  END_IF;
  IF Timer_machining.Q THEN
    Step3 := FALSE; (*reset*)
  END_IF;
  Timer_conveyor(IN := C2_working, PT := T#6000ms);
  IF Timer_conveyor.Q THEN
    C2_working := FALSE; (*reset*)
  END_IF;
  TON4(IN := C2_afterM, PT := T#2000ms);
  IF TON4.Q THEN
    C2_afterM := FALSE; (*reset*)
  END_IF;
  BOOL_TO_DINT41_OUT := BOOL_TO_DINT(EN := TRUE, IN := C2_working, ENO => BOOL_TO_DINT41_ENO);
  C2_working_int := BOOL_TO_DINT41_OUT;
  BOOL_TO_DINT105_OUT := BOOL_TO_DINT(EN := TRUE, IN := C2_afterM, ENO => BOOL_TO_DINT105_ENO);
  C2_afterM_int := BOOL_TO_DINT105_OUT;
  BOOL_TO_DINT51_OUT := BOOL_TO_DINT(EN := TRUE, IN := Step1, ENO => BOOL_TO_DINT51_ENO);
  Step1_int := BOOL_TO_DINT51_OUT;
  BOOL_TO_DINT85_OUT := BOOL_TO_DINT(EN := TRUE, IN := Step2, ENO => BOOL_TO_DINT85_ENO);
  Step2_int := BOOL_TO_DINT85_OUT;
  BOOL_TO_DINT90_OUT := BOOL_TO_DINT(EN := TRUE, IN := Step3, ENO => BOOL_TO_DINT90_ENO);
  Step3_int := BOOL_TO_DINT90_OUT;
  BOOL_TO_DINT95_OUT := BOOL_TO_DINT(EN := TRUE, IN := Pause1, ENO => BOOL_TO_DINT95_ENO);
  Pause1_int := BOOL_TO_DINT95_OUT;
  BOOL_TO_DINT100_OUT := BOOL_TO_DINT(EN := TRUE, IN := Pause2, ENO => BOOL_TO_DINT100_ENO);
  Pause2_int := BOOL_TO_DINT100_OUT;
END_PROGRAM

CONFIGURATION Config0

  RESOURCE Res0 ON PLC
    TASK TaskMain(INTERVAL := T#50ms,PRIORITY := 0);
    PROGRAM Inst0 WITH TaskMain : Cell2;
  END_RESOURCE
END_CONFIGURATION

(* ---- test3.st ---- *)
PROGRAM Cell3
  VAR
    C2_IR AT %IX0.3 : BOOL := true;
    M2_IR AT %IX0.4 : BOOL := true;
    Main AT %IX0.6 : BOOL := true;
    M2_motor AT %QX0.2 : BOOL := true;
    C3_motor AT %QX0.4 : BOOL := true;
  END_VAR
  VAR
    C3_working : BOOL := false;
  END_VAR
  VAR
    C3_working_int AT %MD1 : DINT := 0;
  END_VAR
  VAR
    C3_afterM : BOOL := false;
  END_VAR
  VAR
    C3_afterM_int AT %MD2 : DINT := 0;
  END_VAR
  VAR
    Step1 : BOOL := false;
  END_VAR
  VAR
    Step1_int AT %MD3 : DINT := 0;
  END_VAR
  VAR
    Step2 : BOOL := false;
  END_VAR
  VAR
    Step2_int AT %MD4 : DINT := 0;
  END_VAR
  VAR
    Pause : BOOL := false;
  END_VAR
  VAR
    Pause_int AT %MD5 : DINT := 0;
  END_VAR
  VAR
    Timer_conveyor : TON;
    Timer_machining : TON;
    TON0 : TON;
    TON1 : TON;
    TON2 : TON;
    TON3 : TON;
    C2_IR_working : BOOL := false;
    BOOL_TO_DINT70_ENO : BOOL;
    BOOL_TO_DINT70_OUT : DINT;
    BOOL_TO_DINT41_ENO : BOOL;
    BOOL_TO_DINT41_OUT : DINT;
    BOOL_TO_DINT51_ENO : BOOL;
    BOOL_TO_DINT51_OUT : DINT;
    BOOL_TO_DINT75_ENO : BOOL;
    BOOL_TO_DINT75_OUT : DINT;
    BOOL_TO_DINT80_ENO : BOOL;
    BOOL_TO_DINT80_OUT : DINT;
  END_VAR

  IF NOT(C2_IR) THEN
    C2_IR_working := TRUE; (*set*)
  END_IF;
  IF C2_IR AND C2_IR_working THEN
    C3_working := TRUE; (*set*)
  END_IF;
  C3_motor := NOT((C3_afterM OR C3_working) AND NOT(Main));
  IF NOT(M2_IR) AND C3_working THEN
    Step1 := TRUE; (*set*)
  END_IF;
  IF NOT(M2_IR) AND C3_working THEN
    C2_IR_working := FALSE; (*reset*)
  END_IF;
  IF NOT(M2_IR) AND C3_working THEN
    C3_working := FALSE; (*reset*)
  END_IF;
  M2_motor := NOT((Step1 OR Step2) AND NOT(Main));
  Timer_machining(IN := Step1, PT := T#2000ms);
  IF Timer_machining.Q THEN
    Pause := TRUE; (*set*)
  END_IF;
  IF Timer_machining.Q THEN
    Step1 := FALSE; (*reset*)
  END_IF;
  TON2(IN := Pause, PT := T#1000ms);
  IF TON2.Q THEN
    Step2 := TRUE; (*set*)
  END_IF;
  IF TON2.Q THEN
    Pause := FALSE; (*reset*)
  END_IF;
  TON1(IN := Step2, PT := T#2000ms);
  IF TON1.Q THEN
    C3_afterM := TRUE; (*set*)
  END_IF;
  IF TON1.Q THEN
    Step2 := FALSE; (*reset*)
  END_IF;
  Timer_conveyor(PT := T#6000ms);
  IF Timer_conveyor.Q THEN
    C3_working := FALSE; (*reset*)
  END_IF;
  TON3(IN := C3_afterM, PT := T#2000ms);
  IF TON3.Q THEN
    C3_afterM := FALSE; (*reset*)
  END_IF;
  BOOL_TO_DINT70_OUT := BOOL_TO_DINT(EN := TRUE, IN := C3_working, ENO => BOOL_TO_DINT70_ENO);
  C3_working_int := BOOL_TO_DINT70_OUT;
  BOOL_TO_DINT41_OUT := BOOL_TO_DINT(EN := TRUE, IN := C3_afterM, ENO => BOOL_TO_DINT41_ENO);
  C3_afterM_int := BOOL_TO_DINT41_OUT;
  BOOL_TO_DINT51_OUT := BOOL_TO_DINT(EN := TRUE, IN := Step1, ENO => BOOL_TO_DINT51_ENO);
  Step1_int := BOOL_TO_DINT51_OUT;
  BOOL_TO_DINT75_OUT := BOOL_TO_DINT(EN := TRUE, IN := Step2, ENO => BOOL_TO_DINT75_ENO);
  Step2_int := BOOL_TO_DINT75_OUT;
  BOOL_TO_DINT80_OUT := BOOL_TO_DINT(EN := TRUE, IN := Pause, ENO => BOOL_TO_DINT80_ENO);
  Pause_int := BOOL_TO_DINT80_OUT;
  TON0(IN := NOT(C2_IR));
END_PROGRAM

CONFIGURATION Config0

  RESOURCE Res0 ON PLC
    TASK TaskMain(INTERVAL := T#50ms,PRIORITY := 0);
    PROGRAM Inst0 WITH TaskMain : Cell3;
  END_RESOURCE
END_CONFIGURATION

(* ---- test4.st ---- *)
PROGRAM Cell4
  VAR
    R2_front AT %IX0.2 : BOOL := true;
  END_VAR
  VAR
    C3_IR_working : BOOL := false;
  END_VAR
  VAR
    R2_rear AT %IX0.3 : BOOL := true;
    C4_endIR AT %IX0.4 : BOOL := true;
    C3_IR AT %IX0.5 : BOOL := true;
    Main AT %IX0.6 : BOOL := false;
    R2_fwd_motor AT %QX0.2 : BOOL := true;
    R2_bwd_motor AT %QX0.3 : BOOL := true;
    C4_motor AT %QX0.4 : BOOL := true;
  END_VAR
  VAR
    C4_working : BOOL := false;
  END_VAR
  VAR
    C4_working_int AT %MD1 : DINT := 0;
  END_VAR
  VAR
    R2_in_transit : BOOL := false;
  END_VAR
  VAR
    R2_in_transit_int AT %MD3 : DINT := 0;
  END_VAR
  VAR
    R2_fwd : BOOL := false;
  END_VAR
  VAR
    R2_fwd_int AT %MD4 : DINT := 0;
  END_VAR
  VAR
    R2_bwd : BOOL := false;
  END_VAR
  VAR
    R2_bwd_int AT %MD5 : DINT := 0;
  END_VAR
  VAR
    Timer_in_transit : TON;
    BOOL_TO_DINT49_ENO : BOOL;
    BOOL_TO_DINT49_OUT : DINT;
    BOOL_TO_DINT64_ENO : BOOL;
    BOOL_TO_DINT64_OUT : DINT;
    BOOL_TO_DINT61_ENO : BOOL;
    BOOL_TO_DINT61_OUT : DINT;
    BOOL_TO_DINT67_ENO : BOOL;
    BOOL_TO_DINT67_OUT : DINT;
  END_VAR

  IF NOT(C3_IR) THEN
    C3_IR_working := TRUE; (*set*)
  END_IF;
  IF C3_IR AND C3_IR_working THEN
    R2_in_transit := TRUE; (*set*)
  END_IF;
  Timer_in_transit(IN := R2_in_transit, PT := T#1000ms);
  IF Timer_in_transit.Q THEN
    R2_fwd := TRUE; (*set*)
  END_IF;
  IF Timer_in_transit.Q THEN
    C4_working := TRUE; (*set*)
  END_IF;
  IF Timer_in_transit.Q THEN
    R2_in_transit := FALSE; (*reset*)
  END_IF;
  R2_fwd_motor := NOT(R2_fwd AND NOT(Main));
  IF Timer_in_transit.Q THEN
    C3_IR_working := FALSE; (*reset*)
  END_IF;
  IF NOT(R2_front) AND R2_fwd THEN
    R2_bwd := TRUE; (*set*)
  END_IF;
  IF NOT(R2_front) AND R2_fwd THEN
    R2_fwd := FALSE; (*reset*)
  END_IF;
  R2_bwd_motor := NOT(R2_bwd AND NOT(Main) AND TRUE);
  IF NOT(R2_rear) AND R2_bwd THEN
    R2_bwd := FALSE; (*reset*)
  END_IF;
  C4_motor := NOT(C4_working AND NOT(Main));
  IF NOT(C4_endIR) AND C4_working THEN
    C4_working := FALSE; (*reset*)
  END_IF;
  BOOL_TO_DINT49_OUT := BOOL_TO_DINT(EN := TRUE, IN := C4_working, ENO => BOOL_TO_DINT49_ENO);
  C4_working_int := BOOL_TO_DINT49_OUT;
  BOOL_TO_DINT64_OUT := BOOL_TO_DINT(EN := TRUE, IN := R2_in_transit, ENO => BOOL_TO_DINT64_ENO);
  R2_in_transit_int := BOOL_TO_DINT64_OUT;
  BOOL_TO_DINT61_OUT := BOOL_TO_DINT(EN := TRUE, IN := R2_fwd, ENO => BOOL_TO_DINT61_ENO);
  R2_fwd_int := BOOL_TO_DINT61_OUT;
  BOOL_TO_DINT67_OUT := BOOL_TO_DINT(EN := TRUE, IN := R2_bwd, ENO => BOOL_TO_DINT67_ENO);
  R2_bwd_int := BOOL_TO_DINT67_OUT;
END_PROGRAM

CONFIGURATION Config0

  RESOURCE Res0 ON PLC
    TASK TaskMain(INTERVAL := T#50ms,PRIORITY := 0);
    PROGRAM Inst0 WITH TaskMain : Cell4;
  END_RESOURCE
END_CONFIGURATION
